FUNCTION_BLOCK SPLIT_AB_INTO_AX (* this Function splits the 8 AX (BOOL) adapters from a AB (BYTE) *)
  (* Standard: 61499-2; Description: Copyright (c) 2026 Meisterschulen am Ostbahnhof SPDX-License-Identifier: EPL-2.0 *)
  (* Version 1.0, 2026-03-05, Franz Höpfinger, Meisterschulen am Ostbahnhof, initial API and implementation and/or initial documentation *)
  PACKAGE adapter::splitting;
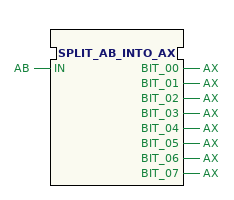
  SOCKETS
    IN : adapter::types::unidirectional::AB; (* BYTE Input *)
  END_SOCKETS
  PLUGS
    BIT_00 : adapter::types::unidirectional::AX; (* Bool Bit 0 *)
    BIT_01 : adapter::types::unidirectional::AX; (* Bool Bit 1 *)
    BIT_02 : adapter::types::unidirectional::AX; (* Bool Bit 2 *)
    BIT_03 : adapter::types::unidirectional::AX; (* Bool Bit 3 *)
    BIT_04 : adapter::types::unidirectional::AX; (* Bool Bit 4 *)
    BIT_05 : adapter::types::unidirectional::AX; (* Bool Bit 5 *)
    BIT_06 : adapter::types::unidirectional::AX; (* Bool Bit 6 *)
    BIT_07 : adapter::types::unidirectional::AX; (* Bool Bit 7 *)
  END_PLUGS
END_FUNCTION_BLOCK
